(* CODESYS project ChainController.library
   Author: Filippo Boido
   Placeholder: ChainController
   Title: ChainController
   Version: 1.0.0.0
   Company: FactoryAutomation

Project tree, tasks and I/O mapping:
  libraries: Tc2_Standard, * (Beckhoff Automation GmbH); Tc2_System, * (Beckhoff Automation GmbH); Tc3_Module, * (Beckhoff Automation GmbH)
  DUTs/
    data type E_ChainStateMachine
    data type ST_ChainDefinition
    data type ST_ChainStateMachine
  GVLs/
    global variables GVL_Constants
  POUs/
    function block FB_Chain [ST]: cmdIgnite, cmdStart, cmdStop, cmdWait, define, getDefinition, getRefChainReleases, getRefReleaseResult, getState, busy, error, init, ready, stop, wait
    function block FB_ChainController [ST]: addChain, releaseCheck, releaseForChain, releaseFromChain, releaseResult
    function block FB_TestChain1 [ST]: init
    function block FB_TestChain2 [ST]: init
    interface I_Chain: getDefinition, getRefChainReleases, getRefReleaseResult
    interface I_ChainController: addChain, releaseForChain, releaseFromChain, releaseResult
    program MAIN [ST]
  Version/
    global variables Global_Version
  VISUs/
*)

// DUTs/E_ChainStateMachine
TYPE E_ChainStateMachine :
(
	eNoState := 0,
	eInit,
	eReady,
	eBusy,
	eStop,
	eWait,
	eError
);
END_TYPE

// DUTs/ST_ChainDefinition
TYPE ST_ChainDefinition :
STRUCT
	uiChainNumber : UINT;
	sChainName : STRING;
END_STRUCT
END_TYPE

// DUTs/ST_ChainStateMachine
TYPE ST_ChainStateMachine :
STRUCT
	bInit : BOOL;
	bReady : BOOL;
	bBusy : BOOL;
	bStop : BOOL;
	bWait : BOOL;
	bError : BOOL;
END_STRUCT
END_TYPE

// GVLs/GVL_Constants

VAR_GLOBAL CONSTANT
	cMaxChains : UINT := 50;
END_VAR

// Version/Global_Version
{attribute 'TcGenerated'}
{attribute 'no-analysis'}
{attribute 'linkalways'}
// This function has been automatically generated from the project information.
VAR_GLOBAL CONSTANT
	{attribute 'const_non_replaced'}
	stLibVersion_ChainController : ST_LibVersion := (iMajor := 1, iMinor := 0, iBuild := 0, iRevision := 0, nFlags := 0, sVersion := '1.0.0.0');
END_VAR

// POUs/FB_Chain
FUNCTION_BLOCK FB_Chain IMPLEMENTS I_Chain
VAR_IN_OUT
	io_fbChainController : FB_ChainController;
END_VAR

VAR
	eChainStateMachine : E_ChainStateMachine;
	uiChainNumber : UINT;
	sChainName : STRING;
	bReleaseResult : BOOL;
	aChainReleases : ARRAY[1..cMaxChains] OF BOOL;

	initStep : UINT;
	readyStep : UINT;
	stopStep : UINT;
	waitStep : UINT;
	busyStep : UINT;
	errorStep : UINT;
	
END_VAR

CASE eChainStateMachine OF

	eNoState:;
	
	eInit:
		init();
	eReady:
		ready();
	eBusy:
		busy();
	eStop:
		stop();
	eWait:
		wait();
	eError:
		error();
	
END_CASE

METHOD cmdIgnite : BOOL
VAR_INPUT
END_VAR
IF eChainStateMachine = eNoState
THEN
	eChainStateMachine := eInit;
END_IF
END_METHOD

METHOD cmdStart : BOOL
VAR_INPUT
END_VAR
eChainStateMachine := eBusy;
END_METHOD

METHOD cmdStop : BOOL
VAR_INPUT
END_VAR
eChainStateMachine := eStop;
END_METHOD

METHOD cmdWait : BOOL
VAR_INPUT
END_VAR
eChainStateMachine := eWait;
END_METHOD

METHOD define : BOOL
VAR_INPUT
	uiChainNumber : UINT;
	sChainName    : STRING;
END_VAR
THIS^.uiChainNumber := uiChainNumber;
THIS^.sChainName := sChainName;
END_METHOD

PROPERTY getDefinition : ST_ChainDefinition
GET
getDefinition.sChainName := sChainName;
getDefinition.uiChainNumber := uiChainNumber;
END_GET
END_PROPERTY

PROPERTY getRefChainReleases : REFERENCE TO ARRAY[1..cMaxChains] OF BOOL
GET
getRefChainReleases REF= aChainReleases;
END_GET
END_PROPERTY

PROPERTY getRefReleaseResult : REFERENCE TO BOOL
GET
getRefReleaseResult REF= bReleaseResult;
END_GET
END_PROPERTY

PROPERTY getState : E_ChainStateMachine
GET
getState := eChainStateMachine;
END_GET
END_PROPERTY

METHOD busy : BOOL
VAR_INPUT
END_VAR
END_METHOD

METHOD error : BOOL
VAR_INPUT
END_VAR
END_METHOD

METHOD init : BOOL
VAR_INPUT
END_VAR
END_METHOD

METHOD ready : BOOL
VAR_INPUT
END_VAR
END_METHOD

METHOD stop : BOOL
VAR_INPUT
END_VAR
END_METHOD

METHOD wait : BOOL
VAR_INPUT
END_VAR
END_METHOD

END_FUNCTION_BLOCK

// POUs/I_Chain
INTERFACE I_Chain

PROPERTY getDefinition : ST_ChainDefinition
GET
END_GET
END_PROPERTY

PROPERTY getRefChainReleases : REFERENCE TO ARRAY[1..cMaxChains] OF BOOL
GET
END_GET
END_PROPERTY

PROPERTY getRefReleaseResult : REFERENCE TO BOOL
GET
END_GET
END_PROPERTY

END_INTERFACE

// POUs/FB_ChainController
FUNCTION_BLOCK FB_ChainController IMPLEMENTS I_ChainController
VAR_INPUT
	
END_VAR
VAR_OUTPUT
END_VAR
VAR
	aChains : ARRAY[1..cMaxChains] OF I_Chain;
	uiNextChain : UINT := 1;
END_VAR

METHOD addChain : I_ChainController 
VAR_INPUT
	itfChain : I_Chain;
END_VAR
VAR
	i: UINT;
END_VAR
addChain := THIS^;

IF itfChain = 0 
OR uiNextChain > cMaxChains 
THEN
	RETURN;
END_IF

//chain already added?
FOR i := 1 TO uiNextChain-1 DO
	IF aChains[i] = itfChain
	THEN
		//yes, already added
		RETURN;
	END_IF
END_FOR

aChains[uiNextChain] := itfChain;
uiNextChain := uiNextChain + 1;
END_METHOD

METHOD releaseCheck : I_ChainController
VAR_INPUT
	itfContractor : I_Chain;
END_VAR
VAR
	i : UINT;
	rReleaseResult :  REFERENCE TO BOOL; 
END_VAR
releaseCheck := THIS^;

FOR i := 1 TO uiNextChain-1 DO
	
	IF itfContractor = aChains[i]
	THEN
		
		rReleaseResult REF= aChains[i].getRefReleaseResult;
		rReleaseResult := TRUE;
		EXIT;
	END_IF
	
END_FOR
END_METHOD

METHOD Public releaseForChain : I_ChainController
VAR_INPUT
	sChainToRelease : STRING;
	itfCommissioner : I_Chain;
END_VAR
VAR
	i : UINT;
	j: UINT;
	stChainDefinition : ST_ChainDefinition; 
	aChainReleases : REFERENCE TO ARRAY[1..cMaxChains] OF BOOL;
END_VAR
releaseForChain := THIS^;

//search for the chain to release
FOR i := 1 TO uiNextChain-1 DO
	stChainDefinition := aChains[i].GetDefinition;
	IF  stChainDefinition.sChainName = sChainToRelease
	THEN
		aChainReleases REF= aChains[i].getRefChainReleases;
		//search for the commissioner
		FOR j := 1 TO uiNextChain-1 DO
			IF aChains[j] = itfCommissioner
			THEN
				aChainReleases[j] := TRUE;
			END_IF
		END_FOR
			
	END_IF
END_FOR
END_METHOD

METHOD Public releaseFromChain : I_ChainController
VAR_INPUT
	sChainReleasing : STRING;
	itfContractor : I_Chain;
END_VAR
VAR
	i : UINT;
	j: UINT;
	stChainDefinition : ST_ChainDefinition; 
	aChainReleases : REFERENCE TO ARRAY[1..cMaxChains] OF BOOL;
	rReleaseResult : REFERENCE TO BOOL; 
END_VAR
releaseFromChain := THIS^;

//search for the contractor
FOR i := 1 TO uiNextChain-1 DO
	
	IF itfContractor = aChains[i]
	THEN
		aChainReleases REF= aChains[i].getRefChainReleases;
		rReleaseResult REF= aChains[i].getRefReleaseResult;
		FOR j := 1 TO uiNextChain-1 DO
			stChainDefinition := aChains[j].getDefinition;
			IF stChainDefinition.sChainName = sChainReleasing
			THEN
				rReleaseResult := rReleaseResult AND aChainReleases[j]; 
			END_IF
			
		END_FOR
		
	END_IF
	
END_FOR
END_METHOD

METHOD releaseResult : Bool
VAR_INPUT
	itfRequester : I_Chain;
END_VAR
VAR
	i,j : UINT;
	rReleaseResult : REFERENCE TO BOOL; 
	aChainReleases : REFERENCE TO ARRAY[1..cMaxChains] OF BOOL;
END_VAR
FOR i := 1 TO cMaxChains DO
	
	IF  itfRequester = aChains[i]
	THEN
		IF aChains[i].getRefReleaseResult 
		THEN
			releaseResult := TRUE;
			aChainReleases REF= aChains[i].getRefChainReleases;
			//reset the releases
			FOR j := 1 TO uiNextChain-1 DO
				aChainReleases[j] := FALSE;
			END_FOR
			EXIT;
		END_IF
	END_IF
END_FOR
END_METHOD

END_FUNCTION_BLOCK

// POUs/I_ChainController
INTERFACE I_ChainController

METHOD addChain : I_ChainController 
VAR_INPUT
	itfChain : I_Chain;
END_VAR
END_METHOD

METHOD releaseForChain : I_ChainController
VAR_INPUT
	sChainToRelease : STRING;
	itfCommissioner : I_Chain;
END_VAR
END_METHOD

METHOD releaseFromChain : I_ChainController
VAR_INPUT
	sChainReleasing : STRING;
	itfContractor : I_Chain;
END_VAR
END_METHOD

METHOD releaseResult : Bool
VAR_INPUT
	itfRequester : I_Chain;
END_VAR
END_METHOD

END_INTERFACE

// POUs/FB_TestChain1
FUNCTION_BLOCK FB_TestChain1 EXTENDS FB_Chain
VAR_INPUT
END_VAR
VAR_OUTPUT
END_VAR
VAR
END_VAR

super^(io_fbChainController := io_fbChainController);

METHOD init : BOOL
VAR_INPUT
END_VAR
CASE initStep OF

0:
	IF io_fbChainController
		.releaseCheck(THIS^)
		.releaseFromChain(sChainReleasing := 'fbChain2', THIS^)
		.releaseResult(THIS^) 
	THEN
		initStep := 10;
	END_IF
10:
	;
20:
	;
30:

END_CASE
END_METHOD

END_FUNCTION_BLOCK

// POUs/FB_TestChain2
FUNCTION_BLOCK FB_TestChain2 EXTENDS FB_Chain
VAR_INPUT
END_VAR
VAR_OUTPUT
END_VAR
VAR
END_VAR

super^(io_fbChainController := io_fbChainController);

METHOD init : BOOL
VAR_INPUT
END_VAR
CASE initStep OF
0:

10:
	io_fbChainController.releaseForChain(sChainToRelease := 'fbChain1',THIS^);
	initStep := 20;
20:

30:

END_CASE
END_METHOD

END_FUNCTION_BLOCK

// POUs/MAIN
PROGRAM MAIN
VAR
	step : UINT;
	fbChainController : FB_ChainController;
	fbChain1 : FB_TestChain1;
	fbChain2 : FB_TestChain2;
END_VAR

fbChain1(io_fbChainController := fbChainController);
fbChain2(io_fbChainController := fbChainController);

fbChain1.define(uiChainNumber := 1, sChainName := 'fbChain1');
fbChain2.define(uiChainNumber := 2, sChainname := 'fbChain2');

CASE step OF

	10: 
		fbChainController
			.addChain(fbChain1)
			.addChain(fbChain2);
		
		fbChain1.cmdIgnite();
		fbChain2.cmdIgnite();	
		step := 20;
		
	20:
	
		
END_CASE

END_PROGRAM
